// TIA Portal V16 export
// export: Created 2021-08-30T15:03:14.4518812Z, ExportSetting WithDefaults, DisplayName Totally Integrated Automation Portal, DisplayVersion V16, DisplayName TIA Portal Version Control Interface, DisplayVersion V16, DisplayName TIA Portal Openness, DisplayVersion V16, DisplayName STEP 7 Professional, DisplayVersion V16, DisplayName STEP 7 Safety, DisplayVersion V16, DisplayName WinCC Professional, DisplayVersion V16
TYPE "LQParams"
// This block is AUTO GENERATED - DO NOT MODIFY this block!
// Created by ODK_CodeGenerator version 205.100.101.18
// at Mon August 30 17:02:50 2021
// ********************************************************
// stored: IsFailsafeCompliant false
   STRUCT
      Lr : Array[0..3] of LReal;   // [LQ Controller 1/Gain Lr]:LQ_P.Lr
      Ly : Array[0..9] of LReal;   // [LQ Controller 1/Gain Ly]:LQ_P.Ly
   END_STRUCT;
   // Lr[0] := 0.013106;
   // Lr[1..2] := 0.0;
   // Lr[3] := 3.112673;
   // Ly[0..3] := 0.0;
   // Ly[4] := 0.011684;
   // Ly[5] := 0.0;
   // Ly[6] := 3.8E-05;
   // Ly[7..8] := 0.0;
   // Ly[9] := 3.112673;
END_TYPE
